FUNCTION_BLOCK FB_PresenceDetector
VAR_INPUT
END_VAR
VAR_OUTPUT
	bAllPartsPresent : BOOL;
END_VAR
VAR
	aSensors : ARRAY[1..3] OF FB_Sensor;
	i: INT;
END_VAR

IF aSensors[1].bSignal
 AND aSensors[2].bSignal
 AND aSensors[3].bSignal
THEN
	bAllPartsPresent := TRUE;
ELSE
	bAllPartsPresent :=FALSE;
END_IF

END_FUNCTION_BLOCK

(* stored: Version 1.1.0.1, ProductVersion 3.1.4024.0
   POU FB_PresenceDetector: Id {920e735c-29a1-439c-8f37-f621dfe385b4}, SpecialFunc None *)
